// TIA Portal V17 export
// export: Created 2023-12-05T13:40:24.204862Z, ExportSetting WithDefaults, DisplayName Totally Integrated Automation Portal, DisplayVersion V17, DisplayName TIA Portal Openness, DisplayVersion V17, DisplayName TIA Portal Version Control Interface, DisplayVersion V17, DisplayName SINAMICS Startdrive Advanced, DisplayVersion V17, DisplayName SINAMICS Startdrive G130, G150, S120, S150, SINAMICS MV, S210, DisplayVersion V17, DisplayName SINAMICS Startdrive G110M, G120, G120C, G120D, G120P, G115D, DisplayVersion V17, DisplayName STEP 7 Professional, DisplayVersion V17, DisplayName STEP 7 Safety, DisplayVersion V17, DisplayName WinCC Professional, DisplayVersion V17
DATA_BLOCK "DB412 Cycle timers"   // DB412
{ S7_Optimized_Access := 'TRUE' }
VERSION : 0.1
// stored: AutoNumber false, DBAccessibleFromOPCUA true, DBAccessibleFromWebserver true, IsOnlyStoredInLoadMemory false, IsRetainMemResEnabled false, IsWriteProtectedInAS false, MemoryReserve 100
   VAR RETAIN
      ST1 { S7_SetPoint := 'True'} : "St timers";
      ST2 { S7_SetPoint := 'True'} : "St timers";
      "ST1 life time" { S7_SetPoint := 'True'} : "St Life time";
      "ST2 life time" { S7_SetPoint := 'True'} : "St Life time";
      "Machine life time" { S7_SetPoint := 'True'} : "Machine Life time";
   END_VAR
BEGIN
   // ST1.Station.Units[1] : ST1OP02_CUT_NIPPLE
   // ST1.Station.Units[2] : ST1OP03_CUT_FTPS_BRACKET
   // ST1.Station.Units[3] : ST1OP05_WELD_NIPPLE
   // ST1.Station.Units[4] : ST1OP07_WELD_REAR_BRACKET
   // ST1.Station.Units[5] : ST1OP09_WELD_TOP_BRACKET
   // ST1.Station.Units[6] : ST1OP11_WELD_1W_CLIP
   // ST1.Station.Units[7] : ST1OP12_WELD_HARPOON_CLIP
   // ST1.Station.Units[8] : ST1OP13_WELD_GF_FILTER_BRACKET
   // ST1.Station.Units[9] : ST1OP14_WELD_FORT_BOYARD_CLIP
   // ST1.Station.Units[10] : ST1OP15_WELD_RIGHT_BRACKET
   // ST2.Station.Units[1] : ST2OP04_WELD_FILLER_PIPE
   // ST2.Station.Units[2] : ST2OP05_INSERTION
   // ST2.Station.Units[3] : ST2OP06_WELD_FTPS_BRACKET
   // ST2.Station.Units[4] : ST2OP08_WELD_REAR_BRACKET
   // ST2.Station.Units[5] : ST2OP14_WELD_BOSS_1
   // ST2.Station.Units[6] : ST2OP15_WELD_BOSS_2
   // ST2.Station.Units[7] : ST2OP17_OILING_&_FTTPS_ASSY
   // ST2.Station.Units[8] : ST2OP18_PUNCHING
END_DATA_BLOCK
